TYPE ST_MasterStatus_2 :
STRUCT
END_STRUCT
END_TYPE

(* stored: Version 1.1.0.1, ProductVersion 3.1.4024.12
   DUT ST_MasterStatus_2: Id {7bd59fbb-144d-42fe-8b6b-0a98a066f007} *)
